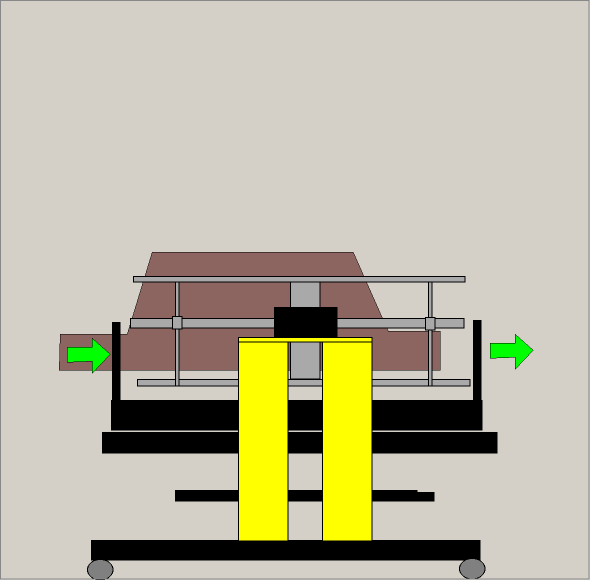
VISUALIZATION studsInScreen  // 590x580
    Polygon (59,370) (60,334) (127,334) (152,252) (353,252) (388,331) (440,331) (440,369) (440,370)
    Rectangle (111,400 371x30)
    Rectangle (256,315 98x30), angle 90
    Rectangle (137,379 333x7)
    Rectangle (175,490 242x11), angle 25
    Rectangle (191,492 243x9), angle 336
    Rectangle (102,432 395x21)
    Rectangle (91,540 389x20)
    Rectangle (238,341 50x200)
    Rectangle (322,341 50x200)
    Ellipse (459,558 26x21)
    Ellipse (87,559 26x21)
    Rectangle (238,337 134x5)
    Rectangle (428,281 4x105)
    Rectangle (175,281 4x105)
    Rectangle (133,276 332x6)
    Rectangle (130,318 334x10)
    Rectangle (425,317 10x13)
    Rectangle (172,316 10x13)
    Rectangle (274,307 63x30)
    Rectangle (473,320 8x101)
    Rectangle (112,322 8x101)
    Polygon (67,357) (67,362) (92,361) (92,373) (110,354) (92,338) (92,347) (67,347)
    Polygon (490,353) (490,358) (515,357) (515,369) (533,350) (515,334) (515,343) (490,343)
END_VISUALIZATION

(* stored: Version 1.1.0.1, ProductVersion 3.1.4024.13
   Visu studsInScreen: Id {8f609e88-8819-4cb6-ba0c-487658ad5433} *)
